// TwinCAT 3 PLC project LargeSortingConveyor
// ProgramVersion: 3.1.4026.11
// libraries:
//   Tc2_Standard, * (Beckhoff Automation GmbH)
//   Tc2_System, * (Beckhoff Automation GmbH)
//   [Resi4MPM], * (Jan Wilch)
//   [xPPU], * (Jan Wilch)
// project tree:
//   / HardwareContainer.TcPOU, MAIN.TcPOU, PlcTask.TcTTO
// (motion and I/O tree: see PLC project crane)
// real-time tasks:
//   TASK PlcTask: cycle T#10ms, priority 20, ADS port 350
//   TASK PlcTask1: cycle T#10ms, priority 23, ADS port 351
//   TASK PlcTask2: cycle T#10ms, priority 22, ADS port 352
//   TASK PlcTask3: cycle T#10ms, priority 21, ADS port 353
// variable links:
//   LargeSortingConveyor/LargeSortingConveyor Instance <-> Device (EtherCAT)/BK2&3 (EK1100)/2&3.11 (EL2004)
//     PlcTask Outputs/MAIN.m_container.m_LSC.Motor.DO_TurnClockwise <-> Channel 4/Output
//     PlcTask Outputs/MAIN.m_container.m_LSC.m_rampPusherMid.DO_Extend <-> Channel 3/Output
//     PlcTask Outputs/MAIN.m_container.m_LSC.m_rampPusherStart.DO_Extend <-> Channel 2/Output
//   LargeSortingConveyor/LargeSortingConveyor Instance <-> Device (EtherCAT)/BK2&3 (EK1100)/2&3.12 (EL2004)
//     PlcTask Outputs/MAIN.m_container.m_LSC.Motor.DO_TurnCounterclockwise <-> Channel 1/Output
//     PlcTask Outputs/MAIN.m_panelMgr.DO_GreenLight <-> Channel 2/Output
//     PlcTask Outputs/MAIN.m_panelMgr.DO_WhiteLight <-> Channel 3/Output
//   LargeSortingConveyor/LargeSortingConveyor Instance <-> Device (EtherCAT)/BK2&3 (EK1100)/2&3.3 (EL1004)
//     PlcTask Inputs/MAIN.m_panelMgr.DI_EStopBtn <-> Channel 3/Input
//     PlcTask Inputs/MAIN.m_panelMgr.DI_StartBtn <-> Channel 4/Input
//   LargeSortingConveyor/LargeSortingConveyor Instance <-> Device (EtherCAT)/BK2&3 (EK1100)/2&3.4 (EL1004)
//     PlcTask Inputs/MAIN.m_container.m_LSC.m_inductiveSensorStart.DI_WPMetallic <-> Channel 4/Input
//     PlcTask Inputs/MAIN.m_container.m_LSC.m_opticalSensorStart.DI_WPLight <-> Channel 2/Input
//     PlcTask Inputs/MAIN.m_container.m_LSC.m_presenceSensorStart.DI_WPDetected <-> Channel 3/Input
//     PlcTask Inputs/MAIN.m_panelMgr.DI_ModeSwitch <-> Channel 1/Input
//   LargeSortingConveyor/LargeSortingConveyor Instance <-> Device (EtherCAT)/BK2&3 (EK1100)/2&3.5 (EL1004)
//     PlcTask Inputs/MAIN.m_container.m_LSC.m_inductiveSensorMid.DI_WPMetallic <-> Channel 2/Input
//     PlcTask Inputs/MAIN.m_container.m_LSC.m_opticalSensorEnd.DI_WPLight <-> Channel 3/Input
//     PlcTask Inputs/MAIN.m_container.m_LSC.m_opticalSensorMid.DI_WPLight <-> Channel 1/Input
//   LargeSortingConveyor/LargeSortingConveyor Instance <-> Device (EtherCAT)/BK2&3 (EK1100)/2&3.6 (EL1004)
//     PlcTask Inputs/MAIN.m_container.m_LSC.m_rampPusherMid.DI_Extended <-> Channel 3/Input
//     PlcTask Inputs/MAIN.m_container.m_LSC.m_rampPusherMid.DI_Retracted <-> Channel 4/Input
//     PlcTask Inputs/MAIN.m_container.m_LSC.m_rampPusherStart.DI_Extended <-> Channel 1/Input
//     PlcTask Inputs/MAIN.m_container.m_LSC.m_rampPusherStart.DI_Retracted <-> Channel 2/Input
//   LargeSortingConveyor/LargeSortingConveyor Instance <-> Device (EtherCAT)/BK4 (EK1100)/4.2 (EL1808)
//     PlcTask Inputs/MAIN.m_container.m_LSC.m_rampEnd.m_presenceSensorRampFull.DI_WPDetected <-> Channel 8/Input
//     PlcTask Inputs/MAIN.m_container.m_LSC.m_rampMiddle.m_presenceSensorRampFull.DI_WPDetected <-> Channel 7/Input
//     PlcTask Inputs/MAIN.m_container.m_LSC.m_rampStart.m_presenceSensorRampFull.DI_WPDetected <-> Channel 6/Input
//   LargeSortingConveyor/LargeSortingConveyor Instance <-> Device (EtherCAT)/BK4 (EK1100)/Term 90 (EL3058)
//     PlcTask Inputs/MAIN.m_container.m_LSC.m_rampPusherMid.AI_PositionTransmitter <-> AI Standard Channel 5/Value
//     PlcTask Inputs/MAIN.m_container.m_LSC.m_rampPusherStart.AI_PositionTransmitter <-> AI Standard Channel 6/Value
//   LargeSortingConveyor/LargeSortingConveyor Instance <-> Device (EtherCAT)/BK7 (EK1100)/7.2 (EL1004)
//     PlcTask Inputs/MAIN.m_container.m_LSC.m_Switch.DI_Extended <-> Channel 4/Input
//     PlcTask Inputs/MAIN.m_container.m_LSC.m_Switch.DI_Retracted <-> Channel 3/Input
//   LargeSortingConveyor/LargeSortingConveyor Instance <-> Device (EtherCAT)/BK7 (EK1100)/7.5 (EL2004)
//     PlcTask Outputs/MAIN.m_container.m_LSC.m_Switch.DO_Extend <-> Channel 3/Output

CONFIGURATION LargeSortingConveyor
    RESOURCE PLC ON TwinCAT3
        TASK PlcTask(INTERVAL := T#10ms, PRIORITY := 20);
        PROGRAM MAIN WITH PlcTask : MAIN;
    END_RESOURCE
END_CONFIGURATION

// ---- MAIN.TcPOU
PROGRAM MAIN
VAR CONSTANT
	IGNORE_DEFINITION: BOOL := TRUE;
END_VAR
VAR
	m_errorManager: ErrorManager;
	m_services: ServiceContainer(ADR(m_errorManager));
	
	m_panelMgr: PanelManager(
		m_services.PtrStateTracker,
		EProcessVariables.Pnl_LSC_Start,
		0,
		EProcessVariables.Pnl_LSC_Mode,
		EProcessVariables.Pnl_LSC_EStop,
		0);
	
	// instantiate machine behavior model
	m_container: HardwareContainer(
		m_services.PtrStateTracker, 
		m_services.PtrProcessManager, 
		ADR(m_errorManager));
	
	m_modes: MachineModes(ADR(m_services), ADR(m_panelMgr));
	
	m_appObservation: ARRAY[EProcessVariables.OpMode_LSC..EProcessVariables.OpMode_LSC] OF SValue;
	
	// TESTING
// 	m_lscConnected: BOOL;
// 	m_craneConnected: BOOL;
// 	m_stackConnected: BOOL;
// 	m_stampConnected: BOOL;
END_VAR

// process state observation
m_appObservation[EProcessVariables.OpMode_LSC].DataType := EDataType.string_t;
m_appObservation[EProcessVariables.OpMode_LSC].Value.String_t := m_modes.SFCCurrentStep;
m_appObservation[EProcessVariables.OpMode_LSC].Defined := TRUE;

// cylic service updates
m_services.PtrStateTracker^.CyclicUpdateStatus(IGNORE_DEFINITION, m_appObservation);
m_services.PtrProcessManager^.CyclicManageBehavior();

// main state machine
m_modes();

// TESTING
// IF m_services.PtrStateTracker^.GetString(EProcessVariables.OpMode_LSC) <> '' THEN
// 	m_lscConnected := TRUE;
// END_IF
// IF m_services.PtrStateTracker^.GetString(EProcessVariables.OpMode_Stack) <> '' THEN
// 	m_stackConnected := TRUE;
// END_IF
// IF m_services.PtrStateTracker^.GetString(EProcessVariables.OpMode_Stamp) <> '' THEN
// 	m_stampConnected := TRUE;
// END_IF
// IF m_services.PtrStateTracker^.GetString(EProcessVariables.OpMode_Crane) <> '' THEN
// 	m_craneConnected := TRUE;
// END_IF

END_PROGRAM

// ---- HardwareContainer.TcPOU
FUNCTION_BLOCK HardwareContainer
VAR_INPUT
END_VAR
VAR_OUTPUT
END_VAR
VAR
	// hardware control POUs
	m_LSC: LargeSortingConveyor;
	m_indic: ActivityIndicator(i_signalProcVar := EProcessVariables.Test_LSCFree);
	
	// products
	{attribute 'OPC.UA.DA' := '1'}
	{attribute 'OPC.UA.DA.Access' := '1'}
	m_LSCWP: xPPUProduct(EProcessVariables.LSC_ProductType, EProcessVariables.LSC_ProductStamped);
	
	// hardware observation (if not included in hardware control)
	m_observeLSC: ObserveLSC(ADR(m_LSC), ADR(m_LSCWP));
	
	// control primitives
	m_LSCTransferWPToRampStart: LSC_TransferWorkpieceTo_RampStart(ADR(m_LSC));
	m_LSCTransferWPToRampMid: LSC_TransferWorkpieceTo_RampMid(ADR(m_LSC));
	m_LSCTransferWPToRampEnd: LSC_TransferWorkpieceTo_RampEnd(ADR(m_LSC));
// 	m_LSCTransferWPToPAC: LSC_TransferWorkpieceTo_PAC(ADR(m_LSC));
	m_LSCSearchWorkpiece: LSC_SearchWorkpiece(ADR(m_LSC));
	
	m_delay: Delay;
	m_indicCP_LSC: IndicateActivity(i_id := EPrimitives.Gen_IndicateActive_LSC, i_ptrIndicator := ADR(m_indic));
	m_forceVal_LSC: ForceProcessVariable(i_id := EPrimitives.Gen_ForceVariable_LSC);
	
	// module sequences
END_VAR

METHOD FB_init : BOOL
VAR_INPUT
	bInitRetains : BOOL; // if TRUE, the retain variables are initialized (warm start / cold start)
	bInCopyCode : BOOL;  // if TRUE, the instance afterwards gets moved into the copy code (online change)

	i_ptrStateTracker: POINTER TO StateTracker;
	i_ptrProcessManager: POINTER TO ProcessManager;
	
	i_ptrErrorManager: POINTER TO ErrorManagerBase;
END_VAR
// provide Services to Behaviors
m_LSCTransferWPToRampStart.ProvideServices(i_ptrProcessManager, i_ptrStateTracker);
m_LSCTransferWPToRampMid.ProvideServices(i_ptrProcessManager, i_ptrStateTracker);
m_LSCTransferWPToRampEnd.ProvideServices(i_ptrProcessManager, i_ptrStateTracker);
// m_LSCTransferWPToPAC.ProvideServices(i_ptrProcessManager, i_ptrStateTracker);
m_LSCSearchWorkpiece.ProvideServices(i_ptrProcessManager, i_ptrStateTracker);

m_delay.ProvideServices(i_ptrProcessManager, i_ptrStateTracker);
m_indicCP_LSC.ProvideServices(i_ptrProcessManager, i_ptrStateTracker);
m_forceVal_LSC.ProvideServices(i_ptrProcessManager, i_ptrStateTracker);

// provide Behaviors to the Process Manager
i_ptrProcessManager^.AddPrimitive(ADR(m_LSCTransferWPToRampStart));
i_ptrProcessManager^.AddPrimitive(ADR(m_LSCTransferWPToRampMid));
i_ptrProcessManager^.AddPrimitive(ADR(m_LSCTransferWPToRampEnd));
// i_ptrProcessManager^.AddPrimitive(ADR(m_LSCTransferWPToPAC));
i_ptrProcessManager^.AddPrimitive(ADR(m_LSCSearchWorkpiece));

i_ptrProcessManager^.AddPrimitive(ADR(m_delay));
i_ptrProcessManager^.AddPrimitive(ADR(m_indicCP_LSC));
i_ptrProcessManager^.AddPrimitive(ADR(m_forceVal_LSC));

// provide observations to the Process Manager
i_ptrStateTracker^.AddObservation(ADR(m_observeLSC));
i_ptrStateTracker^.AddObservation(ADR(m_indic));

// provide workpieces to the Process Manager
i_ptrStateTracker^.RegisterLocalProduct(EProducts.LSC_product, ADR(m_LSCWP));
END_METHOD

END_FUNCTION_BLOCK
